{attribute 'call_after_init'}
FUNCTION_BLOCK FB_evRangeCalculator_Test EXTENDS FB_TestSuite
VAR_INPUT
END_VAR
VAR_OUTPUT
END_VAR
VAR
END_VAR

BasicFunction();

METHOD BasicFunction
VAR_INPUT
END_VAR
VAR
	LastWord : WORD := 2#0000_0000_0000_0010;
END_VAR
TEST('CheckRanges');
//Upper limit equal
AssertTrue(
	F_eVRangeCalculator(300, 0) = 2#0000_0000_0000_0110,
	'Upper limit not inclusive');
//Lower limit equal
AssertTrue(
	F_eVRangeCalculator(300, 0) = 2#0000_0000_0000_0110,
	'Upper limit not inclusive');
//Out of range
AssertFalse(
	F_eVRangeCalculator(300.1, 0) = 2#0000_0000_0000_0100,
	'Out of range failed, whatever you did, it broke this really bad.');
//Negative eV
AssertTrue(
	F_eVRangeCalculator(-300, 0) = 16#FFFF,
	'Working with antimatter? Negative eV should failsafe to FFFF.');	

TEST_FINISHED();

TEST('Check hyst keeps');

AssertTrue(
	F_eVRangeCalculator(350, 2#0000_0000_0000_0010) = 2#0000_0000_0000_0110,
	'Moving up does not stick.');
	
AssertTrue(
	F_eVRangeCalculator(150, 2#0000_0000_0000_0010) = 2#0000_0000_0000_0011,
	'Moving down does not stick.');

TEST_FINISHED();

TEST('Check hyst drops');

AssertTrue(
	F_eVRangeCalculator(351, 2#0000_0000_0000_0010) = 2#0000_0000_0000_0100,
	'Moving up does not drop.');
	
AssertTrue(
	F_eVRangeCalculator(149, 2#0000_0000_0000_0010) = 2#0000_0000_0000_0001,
	'Moving down does not drop.');

TEST_FINISHED();
TEST_FINISHED_NAMED('FOO');
END_METHOD

END_FUNCTION_BLOCK

(* stored: Version 1.1.0.1, ProductVersion 3.1.4024.0
   POU FB_evRangeCalculator_Test: Id {0e192851-333a-0ab1-28cf-f545e9aa8730}, SpecialFunc None
   Method BasicFunction: Id {cf22209d-9899-087d-1556-ffa9f464aec1} *)
